Fanuc KAREL source: kb00101.KL

-- PROVISIONAL review KL for V940-1; original PC SHA256 a38e37e95d1933a7e5375d35443ec4835137c2f0ab8504c66ffa234b7a612321
-- Incomplete behavior may be omitted. Consult companion uncertainty JSON. Do not deploy.
PROGRAM KB00101
%NOLOCKGROUP
BEGIN
  -- V9_ZERO_TABLE_METADATA_HINT layout=0002_ascii; no indexed target words; source/name/runtime held
  -- UNRESOLVED_PC offsets 5-12; opcodes 9D,23
  -- UNRESOLVED_PC offsets 17-26; opcodes 3F,75
  -- UNRESOLVED_PC offsets 31-38; opcodes 9D,23
  -- UNRESOLVED_PC offsets 43-50; opcodes 9D,23
  -- UNRESOLVED_PC offsets 55-62; opcodes 9D,23
  -- UNRESOLVED_PC offsets 67-74; opcodes 9D,23
  -- UNRESOLVED_PC offsets 79-86; opcodes 9D,23
  -- UNRESOLVED_PC offsets 91-98; opcodes 9D,23
  -- UNRESOLVED_PC offsets 103-110; opcodes 9D,23
  -- UNRESOLVED_PC offsets 115-181; opcodes 27,22,22,2A,22,22,22,22,22,22,22,22,31
  -- UNRESOLVED_PC offsets 186-190; opcodes 7F
END KB00101
